(* PLC project C, V P 1 *)
(* stored: creationDateTime 2026-01-01T00:00:00 *)

PROGRAM Rungs

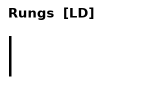
(* LD diagram, written out as Structured Text *)
END_PROGRAM
